INTERFACE I_McAxis

PROPERTY AxisRef : reference to AXIS_REF
GET
END_GET
END_PROPERTY

METHOD Disable : E_PROGRESS
VAR_INPUT
  Execute           : BOOL;
END_VAR
END_METHOD

METHOD Enable : E_PROGRESS
VAR_INPUT
  Execute           : BOOL;
END_VAR
END_METHOD

METHOD Halt : E_PROGRESS
VAR_INPUT
  Execute           : BOOL;
  Dec               : LREAL;
  Jerk              : LREAL;
END_VAR
END_METHOD

PROPERTY Position : LREAL
GET
END_GET
END_PROPERTY

METHOD ReadParameter : E_PROGRESS
VAR_INPUT
  Execute           : BOOL;
  ParameterNumber   : Tc2_MC2.MC_AxisParameter;
END_VAR
END_METHOD

PROPERTY ReadParameterValue : LREAL
GET
END_GET
END_PROPERTY

METHOD Reset : E_PROGRESS
VAR_INPUT
  Execute           : BOOL;
END_VAR
END_METHOD

METHOD Stop : E_PROGRESS
VAR_INPUT
  Execute           : BOOL;
  Dec               : LREAL;
  Jerk              : LREAL;
END_VAR
END_METHOD

METHOD WriteParameter : E_PROGRESS
VAR_INPUT
  Execute           : BOOL;
  Value             : LREAL;
  ParameterNumber   : Tc2_MC2.MC_AxisParameter;
END_VAR
END_METHOD

METHOD WriteParameterPersistent : E_PROGRESS
VAR_INPUT
  Execute           : BOOL;
  Value             : LREAL;
  ParameterNumber   : Tc2_MC2.MC_AxisParameter;
END_VAR
END_METHOD

END_INTERFACE

(* stored: Version 1.1.0.1, ProductVersion 3.1.4026.18
   Itf I_McAxis: Id {df9f672e-6c08-07db-39bc-3fcca419c0c5}
   Folder methods: Id {b49529db-ea8c-01b3-3687-85fa88f4ed08}
   Folder properties: Id {1fd118ac-d3fc-4dba-b1a3-479fd44bd13d}
   Property AxisRef: Id {653615dd-2878-4b72-8d04-079697472efe}
   Get Get: Id {8e4019dc-34f1-4a1f-8b70-5940902e8936}
   Method Disable: Id {6733f6f1-eee7-046b-33ae-7a8adfed7590}
   Method Enable: Id {3268550c-0f61-0793-3744-93a382e3a070}
   Method Halt: Id {a0dc8f7e-08ff-058b-0cd9-6d80a8af16ba}
   Property Position: Id {a08b4e22-77b3-4582-8c00-d0e03499f6f4}
   Get Get: Id {044142a5-1d79-44ea-81e4-7a49c5e5f078}
   Method ReadParameter: Id {89506a67-4c73-45c9-a370-bc249ffe7bb9}
   Property ReadParameterValue: Id {b7f7b90d-c73b-4ac9-b7d8-0512bb3a7546}
   Get Get: Id {3d317b6c-4bb7-4802-af8c-d26bc0ad986d}
   Method Reset: Id {b60d6850-a4c7-07c3-05ec-3f927ae74504}
   Method Stop: Id {9ed3be03-537d-07e4-2377-251305834f1b}
   Method WriteParameter: Id {8fd5a67a-ea90-4314-8d4d-f4e5bfad79c4}
   Method WriteParameterPersistent: Id {ddea80af-6427-4a6e-82a8-634132ea64ed} *)
